(* Logix 5000 project; controller AMP_Servo_Demo vendor 1 type 14 code 154 rev 32.15; software revision 32.05; part 5 of 5 *)
(* tags used below, declared in another part *)
   AMP_Axis1_Absolute_Move_Inst : AMP_Absolute_Move;
   AMP_Axis1_Alarm_Code_Inst : AMP_Alarm_Code;
   AMP_Axis1_Alarm_Reset_Inst : AMP_Alarm_Reset;
   AMP_Axis1_Crash_Stop_Inst : AMP_Crash_Stop;
   AMP_Axis1_DI_Monitor_Inst : AMP_DI_Monitor;
   AMP_Axis1_DO_Control_Inst : AMP_DO_Control;
   AMP_Axis1_Homing_Inst : AMP_Home;
   AMP_Axis1_Inputs : AMP_Input_Assembly_Servo_v2;
   AMP_Axis1_Motor_Disable_Inst : AMP_Motor_Disable;
   AMP_Axis1_Motor_Enable_Inst : AMP_Motor_Enable;
   AMP_Axis1_Motor_Jog_Inst : AMP_Jog_Move;
   AMP_Axis1_Normal_Stop_Inst : AMP_Normal_Stop;
   AMP_Axis1_Point_to_Poinr_IO_Exec : AMP_Point_to_Point_IO;
   AMP_Axis1_Point_to_Point_FC_Exec : AMP_Point_to_Point_FC;
   AMP_Axis1_Q_Segment_Execute_Inst : AMP_Q_Segment_Execute;
   AMP_Axis1_Relative_Move_Inst : AMP_Relative_Move;
   AMP_Axis1_SCL_Inst : AMP_SCL_Command;
   AMP_Axis1_Set_Position_Inst : AMP_Set_Position;
   AMP_Axis1_Status_Code_Inst : AMP_Status_Code;
   AMP_Axis1_Torque_Inst : AMP_Torque_Control;
   AMP_Axis1_Update_Jog_Speed_Inst : AMP_Update_Jog_Speed;
   AMP_Axis2_Absolute_Move_Inst : AMP_Absolute_Move;
   AMP_Axis2_Alarm_Code_Inst : AMP_Alarm_Code;
   AMP_Axis2_Alarm_Reset_Inst : AMP_Alarm_Reset;
   AMP_Axis2_Crash_Stop_Inst : AMP_Crash_Stop;
   AMP_Axis2_DI_Monitor_Inst : AMP_DI_Monitor;
   AMP_Axis2_DO_Control_Inst : AMP_DO_Control;
   AMP_Axis2_Homing_Inst : AMP_Home;
   AMP_Axis2_Inputs : AMP_Input_Assembly_Servo_v2;
   AMP_Axis2_Motor_Disable_Inst : AMP_Motor_Disable;
   AMP_Axis2_Motor_Enable_Inst : AMP_Motor_Enable;
   AMP_Axis2_Motor_Jog_Inst : AMP_Jog_Move;
   AMP_Axis2_Normal_Stop_Inst : AMP_Normal_Stop;
   AMP_Axis2_Point_to_Poinr_IO_Exec : AMP_Point_to_Point_IO;
   AMP_Axis2_Point_to_Point_FC_Exec : AMP_Point_to_Point_FC;
   AMP_Axis2_Q_Segment_Execute_Inst : AMP_Q_Segment_Execute;
   AMP_Axis2_Relative_Move_Inst : AMP_Relative_Move;
   AMP_Axis2_SCL_Inst : AMP_SCL_Command;
   AMP_Axis2_Set_Position_Inst : AMP_Set_Position;
   AMP_Axis2_Status_Code_Inst : AMP_Status_Code;
   AMP_Axis2_Update_Jog_Speed_Inst : AMP_Update_Jog_Speed;
   AMP_Axis2Torque_Inst : AMP_Torque_Control;
   AMP_Input_Axis1_Inst : AMP_Input_Assembly;
   AMP_Input_Axis2_Inst : AMP_Input_Assembly;
(* Explicit_Messages, continued *)

ROUTINE MainRoutine   (* ladder *)
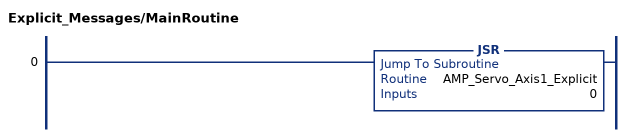
   0: JSR(AMP_Servo_Axis1_Explicit,0);
END_ROUTINE
END_PROGRAM

PROGRAM MainProgram   (* main routine MainRoutine *)

ROUTINE AMP_Servo_Axis1   (* ladder *)
// MDX+ Servo Axis 1 program example using Applied Motion AOIs
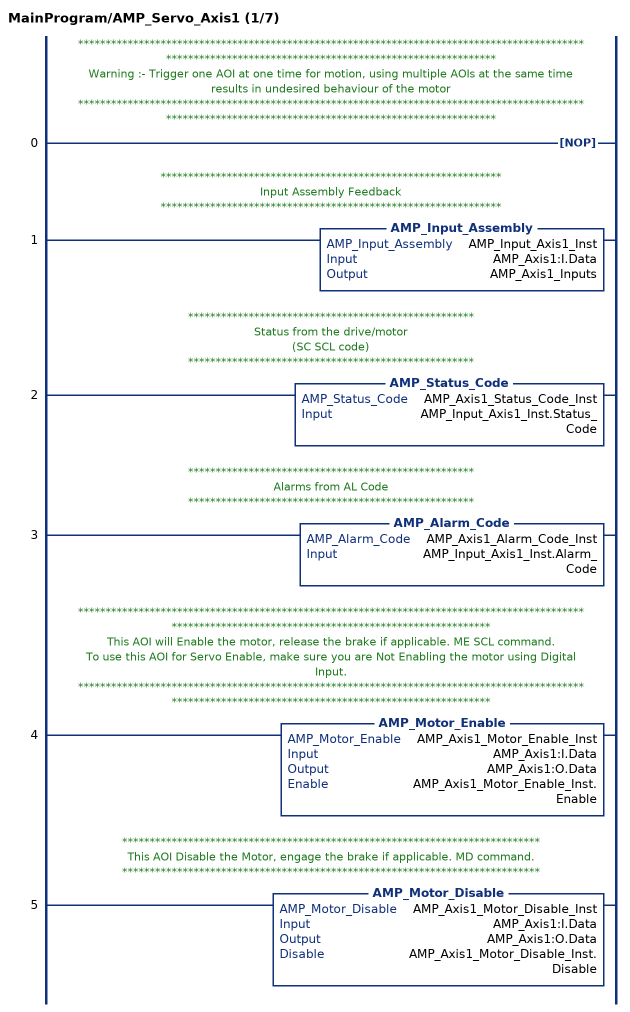
   // ********************************************************************************************************************************************************
   // Warning :- Trigger one AOI at one time for motion, using multiple AOIs at the same time results in undesired behaviour of the motor
   // ********************************************************************************************************************************************************
   0: NOP();
   // **************************************************************
   // Input Assembly Feedback
   // **************************************************************
   1: AMP_Input_Assembly(AMP_Input_Axis1_Inst,AMP_Axis1:I.Data,AMP_Axis1_Inputs);
   // ****************************************************
   // Status from the drive/motor
   // (SC SCL code)
   // ****************************************************
   2: AMP_Status_Code(AMP_Axis1_Status_Code_Inst,AMP_Input_Axis1_Inst.Status_Code);
   // ****************************************************
   //  Alarms from AL Code
   // ****************************************************
   3: AMP_Alarm_Code(AMP_Axis1_Alarm_Code_Inst,AMP_Input_Axis1_Inst.Alarm_Code);
   // ******************************************************************************************************************************************************
   // This AOI will Enable the motor, release the brake if applicable. ME SCL command.
   // To use this AOI for Servo Enable, make sure you are Not Enabling the motor using Digital Input.
   // ******************************************************************************************************************************************************
   4: AMP_Motor_Enable(AMP_Axis1_Motor_Enable_Inst,AMP_Axis1:I.Data,AMP_Axis1:O.Data,AMP_Axis1_Motor_Enable_Inst.Enable);
   // ****************************************************************************
   // This AOI Disable the Motor, engage the brake if applicable. MD command.
   // ****************************************************************************
   5: AMP_Motor_Disable(AMP_Axis1_Motor_Disable_Inst,AMP_Axis1:I.Data,AMP_Axis1:O.Data,AMP_Axis1_Motor_Disable_Inst.Disable);
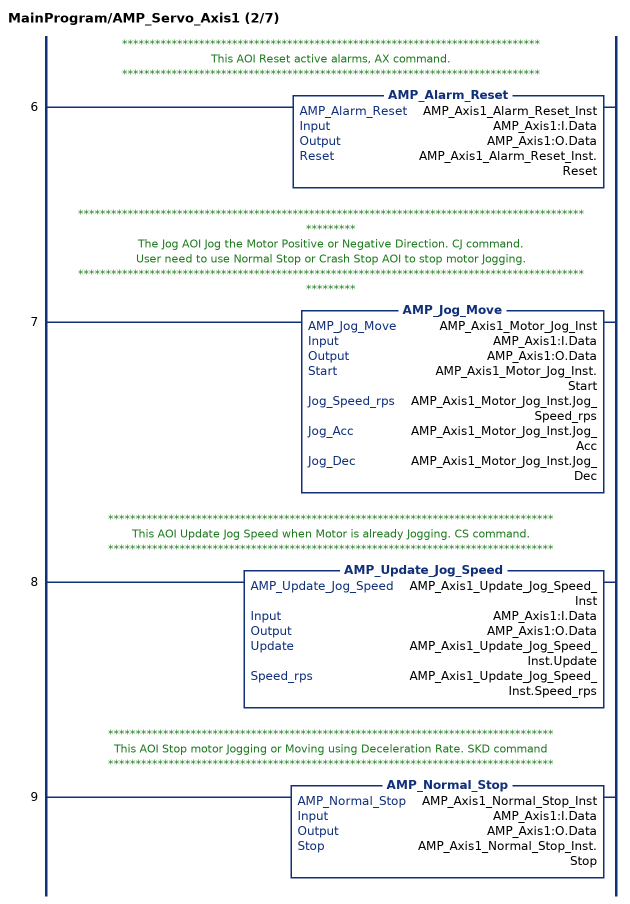
   // ****************************************************************************
   // This AOI Reset active alarms, AX command.
   // ****************************************************************************
   6: AMP_Alarm_Reset(AMP_Axis1_Alarm_Reset_Inst,AMP_Axis1:I.Data,AMP_Axis1:O.Data,AMP_Axis1_Alarm_Reset_Inst.Reset);
   // *****************************************************************************************************
   // The Jog AOI Jog the Motor Positive or Negative Direction. CJ command.
   //  User need to use Normal Stop or Crash Stop AOI to stop motor Jogging.
   // *****************************************************************************************************
   7: AMP_Jog_Move(AMP_Axis1_Motor_Jog_Inst,AMP_Axis1:I.Data,AMP_Axis1:O.Data,AMP_Axis1_Motor_Jog_Inst.Start,AMP_Axis1_Motor_Jog_Inst.Jog_Speed_rps,AMP_Axis1_Motor_Jog_Inst.Jog_Acc,AMP_Axis1_Motor_Jog_Inst.Jog_Dec);
   // *********************************************************************************
   // This AOI Update Jog Speed when Motor is already Jogging. CS command.
   // *********************************************************************************
   8: AMP_Update_Jog_Speed(AMP_Axis1_Update_Jog_Speed_Inst,AMP_Axis1:I.Data,AMP_Axis1:O.Data,AMP_Axis1_Update_Jog_Speed_Inst.Update,AMP_Axis1_Update_Jog_Speed_Inst.Speed_rps);
   // *********************************************************************************
   // This AOI Stop motor Jogging or Moving using Deceleration Rate. SKD command
   // *********************************************************************************
   9: AMP_Normal_Stop(AMP_Axis1_Normal_Stop_Inst,AMP_Axis1:I.Data,AMP_Axis1:O.Data,AMP_Axis1_Normal_Stop_Inst.Stop);
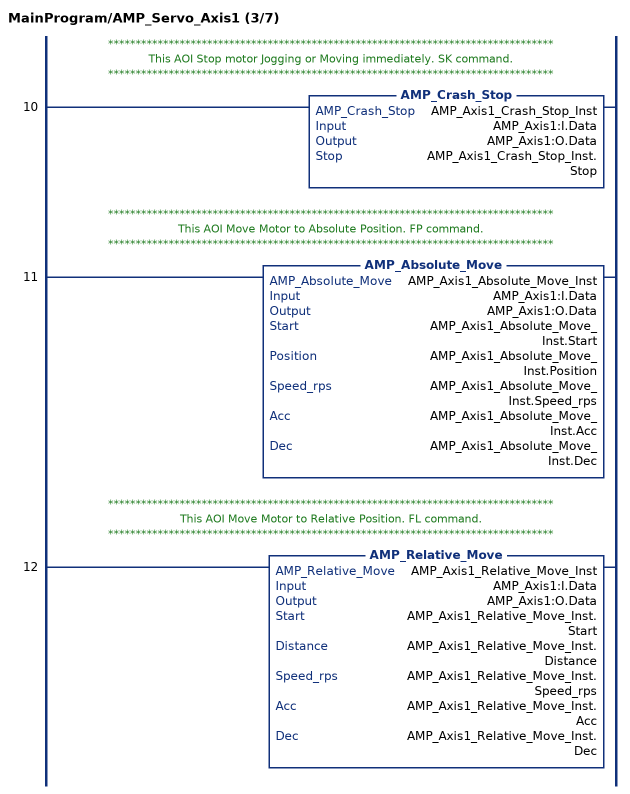
   // *********************************************************************************
   // This AOI Stop motor Jogging or Moving immediately. SK command.
   // *********************************************************************************
   10: AMP_Crash_Stop(AMP_Axis1_Crash_Stop_Inst,AMP_Axis1:I.Data,AMP_Axis1:O.Data,AMP_Axis1_Crash_Stop_Inst.Stop);
   // *********************************************************************************
   // This AOI Move Motor to Absolute Position. FP command.
   // *********************************************************************************
   11: AMP_Absolute_Move(AMP_Axis1_Absolute_Move_Inst,AMP_Axis1:I.Data,AMP_Axis1:O.Data,AMP_Axis1_Absolute_Move_Inst.Start,AMP_Axis1_Absolute_Move_Inst.Position,AMP_Axis1_Absolute_Move_Inst.Speed_rps,AMP_Axis1_Absolute_Move_Inst.Acc,AMP_Axis1_Absolute_Move_Inst.Dec);
   // *********************************************************************************
   // This AOI Move Motor to Relative Position. FL command.
   // *********************************************************************************
   12: AMP_Relative_Move(AMP_Axis1_Relative_Move_Inst,AMP_Axis1:I.Data,AMP_Axis1:O.Data,AMP_Axis1_Relative_Move_Inst.Start,AMP_Axis1_Relative_Move_Inst.Distance,AMP_Axis1_Relative_Move_Inst.Speed_rps,AMP_Axis1_Relative_Move_Inst.Acc,AMP_Axis1_Relative_Move_Inst.Dec);
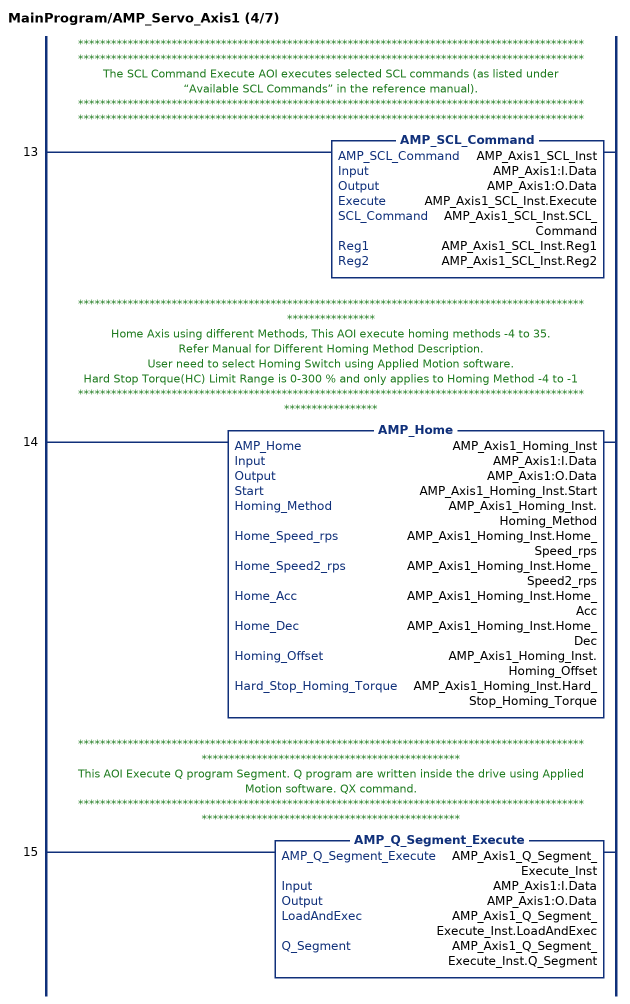
   // ****************************************************************************************************************************************************************************************
   // The SCL Command Execute AOI executes selected SCL commands (as listed under “Available SCL Commands” in the reference manual).
   // ****************************************************************************************************************************************************************************************
   13: AMP_SCL_Command(AMP_Axis1_SCL_Inst,AMP_Axis1:I.Data,AMP_Axis1:O.Data,AMP_Axis1_SCL_Inst.Execute,AMP_Axis1_SCL_Inst.SCL_Command,AMP_Axis1_SCL_Inst.Reg1,AMP_Axis1_SCL_Inst.Reg2);
   // ************************************************************************************************************
   // Home Axis using different Methods, This AOI execute homing methods -4 to 35.
   // Refer Manual for Different Homing Method Description.
   // User need to select Homing Switch using Applied Motion software.
   // Hard Stop Torque(HC) Limit Range is 0-300 % and only applies to Homing Method -4 to -1
   // *************************************************************************************************************
   14: AMP_Home(AMP_Axis1_Homing_Inst,AMP_Axis1:I.Data,AMP_Axis1:O.Data,AMP_Axis1_Homing_Inst.Start,AMP_Axis1_Homing_Inst.Homing_Method,AMP_Axis1_Homing_Inst.Home_Speed_rps,AMP_Axis1_Homing_Inst.Home_Speed2_rps,AMP_Axis1_Homing_Inst.Home_Acc,AMP_Axis1_Homing_Inst.Home_Dec,AMP_Axis1_Homing_Inst.Homing_Offset,AMP_Axis1_Homing_Inst.Hard_Stop_Homing_Torque);
   // *******************************************************************************************************************************************
   // This AOI Execute Q program Segment. Q program are written inside the drive using Applied Motion software. QX command.
   // *******************************************************************************************************************************************
   15: AMP_Q_Segment_Execute(AMP_Axis1_Q_Segment_Execute_Inst,AMP_Axis1:I.Data,AMP_Axis1:O.Data,AMP_Axis1_Q_Segment_Execute_Inst.LoadAndExec,AMP_Axis1_Q_Segment_Execute_Inst.Q_Segment);
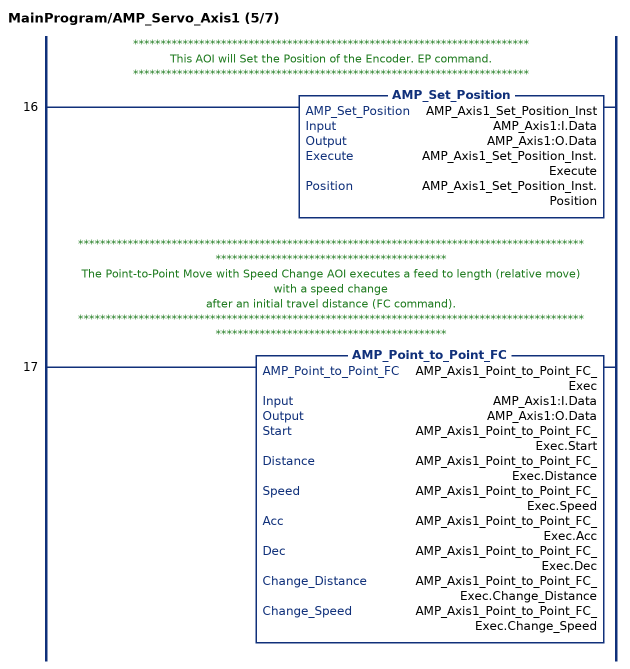
   // ************************************************************************
   // This AOI will Set the Position of the Encoder. EP command.
   // ************************************************************************
   16: AMP_Set_Position(AMP_Axis1_Set_Position_Inst,AMP_Axis1:I.Data,AMP_Axis1:O.Data,AMP_Axis1_Set_Position_Inst.Execute,AMP_Axis1_Set_Position_Inst.Position);
   // **************************************************************************************************************************************
   // The Point-to-Point Move with Speed Change AOI executes a feed to length (relative move) with a speed change
   //  after an initial travel distance (FC command).
   // **************************************************************************************************************************************
   17: AMP_Point_to_Point_FC(AMP_Axis1_Point_to_Point_FC_Exec,AMP_Axis1:I.Data,AMP_Axis1:O.Data,AMP_Axis1_Point_to_Point_FC_Exec.Start,AMP_Axis1_Point_to_Point_FC_Exec.Distance,AMP_Axis1_Point_to_Point_FC_Exec.Speed,AMP_Axis1_Point_to_Point_FC_Exec.Acc,AMP_Axis1_Point_to_Point_FC_Exec.Dec,AMP_Axis1_Point_to_Point_FC_Exec.Change_Distance,AMP_Axis1_Point_to_Point_FC_Exec.Change_Speed);
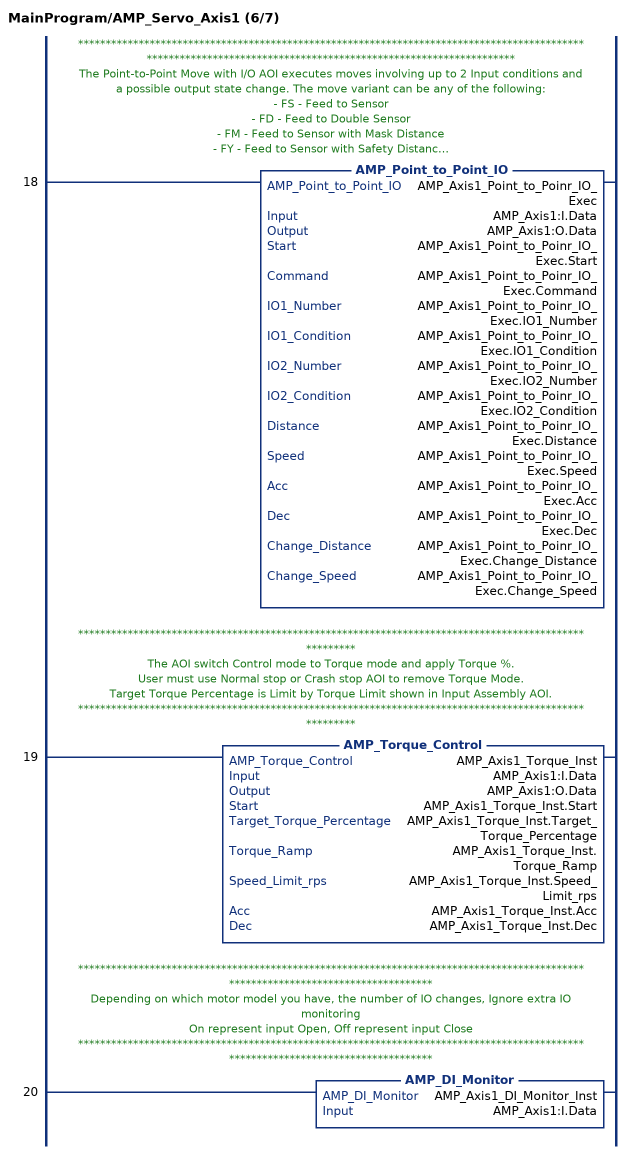
   // ***************************************************************************************************************************************************************
   // The Point-to-Point Move with I/O AOI executes moves involving up to 2 Input conditions and a possible output state change. The move variant can be any of the following:
   // - FS - Feed to Sensor
   // - FD - Feed to Double Sensor
   // - FM - Feed to Sensor with Mask Distance
   // - FY - Feed to Sensor with Safety Distance
   // - FO - Feed to Length and Set Output
   // - SH - Seek Home
   // All six(6) of the above variants need exactly one I/O point except for FD which requires a second I/O point to be specified in the parameters.
   // *************************************************************************************************************************************************************************
   18: AMP_Point_to_Point_IO(AMP_Axis1_Point_to_Poinr_IO_Exec,AMP_Axis1:I.Data,AMP_Axis1:O.Data,AMP_Axis1_Point_to_Poinr_IO_Exec.Start,AMP_Axis1_Point_to_Poinr_IO_Exec.Command,AMP_Axis1_Point_to_Poinr_IO_Exec.IO1_Number,AMP_Axis1_Point_to_Poinr_IO_Exec.IO1_Condition,AMP_Axis1_Point_to_Poinr_IO_Exec.IO2_Number,AMP_Axis1_Point_to_Poinr_IO_Exec.IO2_Condition,AMP_Axis1_Point_to_Poinr_IO_Exec.Distance,AMP_Axis1_Point_to_Poinr_IO_Exec.Speed,AMP_Axis1_Point_to_Poinr_IO_Exec.Acc,AMP_Axis1_Point_to_Poinr_IO_Exec.Dec,AMP_Axis1_Point_to_Poinr_IO_Exec.Change_Distance,AMP_Axis1_Point_to_Poinr_IO_Exec.Change_Speed);
   // *****************************************************************************************************
   // The AOI switch Control mode to Torque mode and apply Torque %.
   // User must use Normal stop or Crash stop AOI to remove Torque Mode.
   // Target Torque Percentage is Limit by Torque Limit shown in Input Assembly AOI.
   // *****************************************************************************************************
   19: AMP_Torque_Control(AMP_Axis1_Torque_Inst,AMP_Axis1:I.Data,AMP_Axis1:O.Data,AMP_Axis1_Torque_Inst.Start,AMP_Axis1_Torque_Inst.Target_Torque_Percentage,AMP_Axis1_Torque_Inst.Torque_Ramp,AMP_Axis1_Torque_Inst.Speed_Limit_rps,AMP_Axis1_Torque_Inst.Acc,AMP_Axis1_Torque_Inst.Dec);
   // *********************************************************************************************************************************
   // Depending on which motor model you have, the number of IO changes, Ignore extra IO monitoring
   // On represent input Open, Off represent input Close
   // *********************************************************************************************************************************
   20: AMP_DI_Monitor(AMP_Axis1_DI_Monitor_Inst,AMP_Axis1:I.Data);
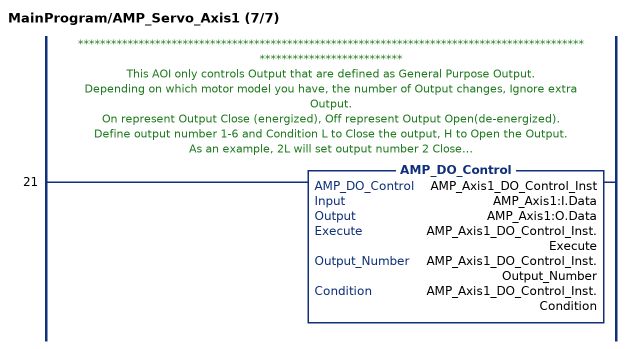
   // **********************************************************************************************************************
   // This AOI only controls Output that are defined as General Purpose Output.
   // Depending on which motor model you have, the number of Output changes, Ignore extra Output.
   // On represent Output Close (energized), Off represent Output Open(de-energized).
   // Define output number 1-6 and Condition L to Close the output, H to Open the Output.
   // As an example, 2L will set output number 2 Close.
   // **********************************************************************************************************************
   21: AMP_DO_Control(AMP_Axis1_DO_Control_Inst,AMP_Axis1:I.Data,AMP_Axis1:O.Data,AMP_Axis1_DO_Control_Inst.Execute,AMP_Axis1_DO_Control_Inst.Output_Number,AMP_Axis1_DO_Control_Inst.Condition);
END_ROUTINE

ROUTINE AMP_Servo_Axis2   (* ladder *)
// M56S Servo Axis 2 program example using Applied Motion AOIs
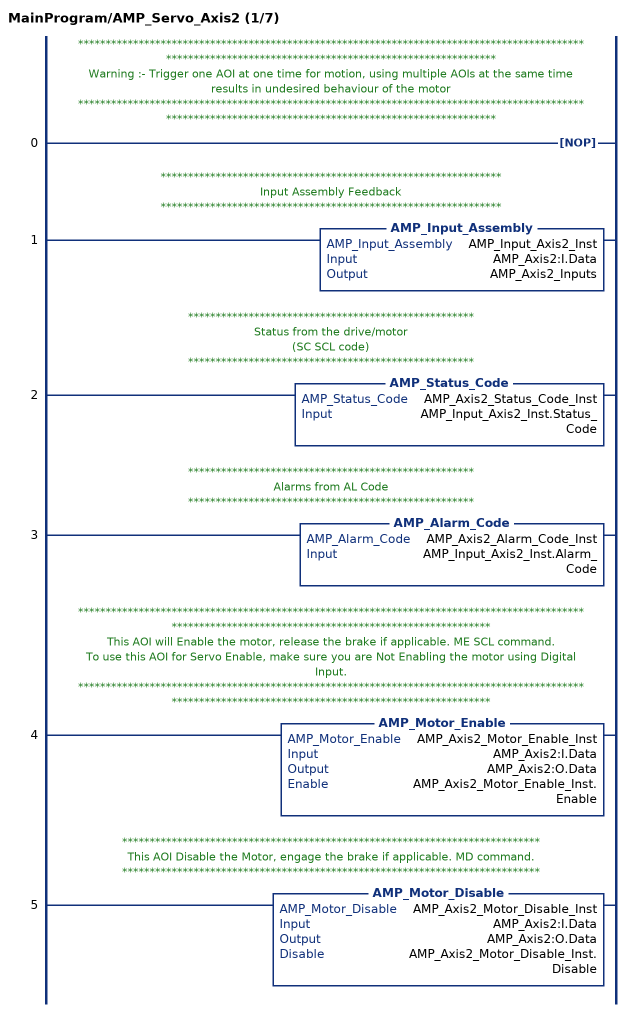
   // ********************************************************************************************************************************************************
   // Warning :- Trigger one AOI at one time for motion, using multiple AOIs at the same time results in undesired behaviour of the motor
   // ********************************************************************************************************************************************************
   0: NOP();
   // **************************************************************
   // Input Assembly Feedback
   // **************************************************************
   1: AMP_Input_Assembly(AMP_Input_Axis2_Inst,AMP_Axis2:I.Data,AMP_Axis2_Inputs);
   // ****************************************************
   // Status from the drive/motor
   // (SC SCL code)
   // ****************************************************
   2: AMP_Status_Code(AMP_Axis2_Status_Code_Inst,AMP_Input_Axis2_Inst.Status_Code);
   // ****************************************************
   //  Alarms from AL Code
   // ****************************************************
   3: AMP_Alarm_Code(AMP_Axis2_Alarm_Code_Inst,AMP_Input_Axis2_Inst.Alarm_Code);
   // ******************************************************************************************************************************************************
   // This AOI will Enable the motor, release the brake if applicable. ME SCL command.
   // To use this AOI for Servo Enable, make sure you are Not Enabling the motor using Digital Input.
   // ******************************************************************************************************************************************************
   4: AMP_Motor_Enable(AMP_Axis2_Motor_Enable_Inst,AMP_Axis2:I.Data,AMP_Axis2:O.Data,AMP_Axis2_Motor_Enable_Inst.Enable);
   // ****************************************************************************
   // This AOI Disable the Motor, engage the brake if applicable. MD command.
   // ****************************************************************************
   5: AMP_Motor_Disable(AMP_Axis2_Motor_Disable_Inst,AMP_Axis2:I.Data,AMP_Axis2:O.Data,AMP_Axis2_Motor_Disable_Inst.Disable);
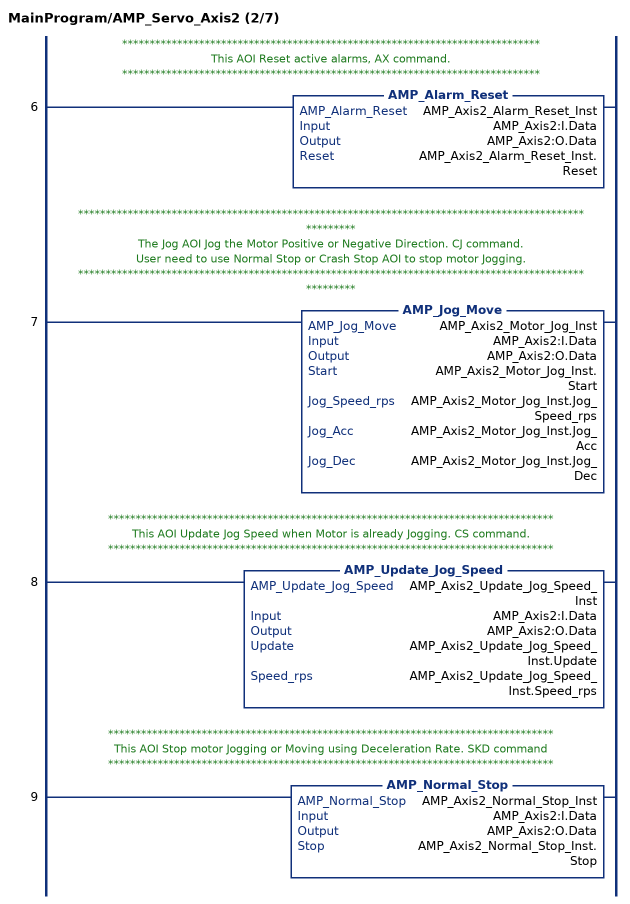
   // ****************************************************************************
   // This AOI Reset active alarms, AX command.
   // ****************************************************************************
   6: AMP_Alarm_Reset(AMP_Axis2_Alarm_Reset_Inst,AMP_Axis2:I.Data,AMP_Axis2:O.Data,AMP_Axis2_Alarm_Reset_Inst.Reset);
   // *****************************************************************************************************
   // The Jog AOI Jog the Motor Positive or Negative Direction. CJ command.
   //  User need to use Normal Stop or Crash Stop AOI to stop motor Jogging.
   // *****************************************************************************************************
   7: AMP_Jog_Move(AMP_Axis2_Motor_Jog_Inst,AMP_Axis2:I.Data,AMP_Axis2:O.Data,AMP_Axis2_Motor_Jog_Inst.Start,AMP_Axis2_Motor_Jog_Inst.Jog_Speed_rps,AMP_Axis2_Motor_Jog_Inst.Jog_Acc,AMP_Axis2_Motor_Jog_Inst.Jog_Dec);
   // *********************************************************************************
   // This AOI Update Jog Speed when Motor is already Jogging. CS command.
   // *********************************************************************************
   8: AMP_Update_Jog_Speed(AMP_Axis2_Update_Jog_Speed_Inst,AMP_Axis2:I.Data,AMP_Axis2:O.Data,AMP_Axis2_Update_Jog_Speed_Inst.Update,AMP_Axis2_Update_Jog_Speed_Inst.Speed_rps);
   // *********************************************************************************
   // This AOI Stop motor Jogging or Moving using Deceleration Rate. SKD command
   // *********************************************************************************
   9: AMP_Normal_Stop(AMP_Axis2_Normal_Stop_Inst,AMP_Axis2:I.Data,AMP_Axis2:O.Data,AMP_Axis2_Normal_Stop_Inst.Stop);
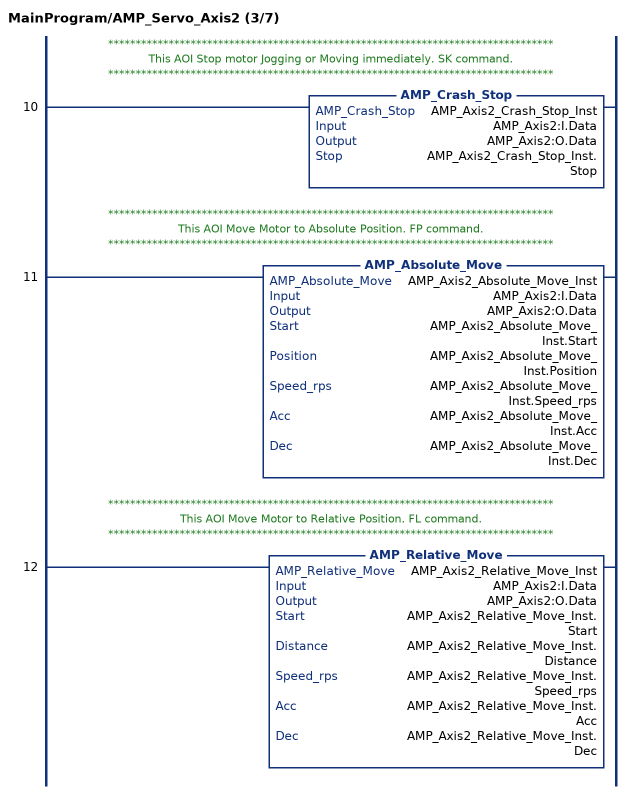
   // *********************************************************************************
   // This AOI Stop motor Jogging or Moving immediately. SK command.
   // *********************************************************************************
   10: AMP_Crash_Stop(AMP_Axis2_Crash_Stop_Inst,AMP_Axis2:I.Data,AMP_Axis2:O.Data,AMP_Axis2_Crash_Stop_Inst.Stop);
   // *********************************************************************************
   // This AOI Move Motor to Absolute Position. FP command.
   // *********************************************************************************
   11: AMP_Absolute_Move(AMP_Axis2_Absolute_Move_Inst,AMP_Axis2:I.Data,AMP_Axis2:O.Data,AMP_Axis2_Absolute_Move_Inst.Start,AMP_Axis2_Absolute_Move_Inst.Position,AMP_Axis2_Absolute_Move_Inst.Speed_rps,AMP_Axis2_Absolute_Move_Inst.Acc,AMP_Axis2_Absolute_Move_Inst.Dec);
   // *********************************************************************************
   // This AOI Move Motor to Relative Position. FL command.
   // *********************************************************************************
   12: AMP_Relative_Move(AMP_Axis2_Relative_Move_Inst,AMP_Axis2:I.Data,AMP_Axis2:O.Data,AMP_Axis2_Relative_Move_Inst.Start,AMP_Axis2_Relative_Move_Inst.Distance,AMP_Axis2_Relative_Move_Inst.Speed_rps,AMP_Axis2_Relative_Move_Inst.Acc,AMP_Axis2_Relative_Move_Inst.Dec);
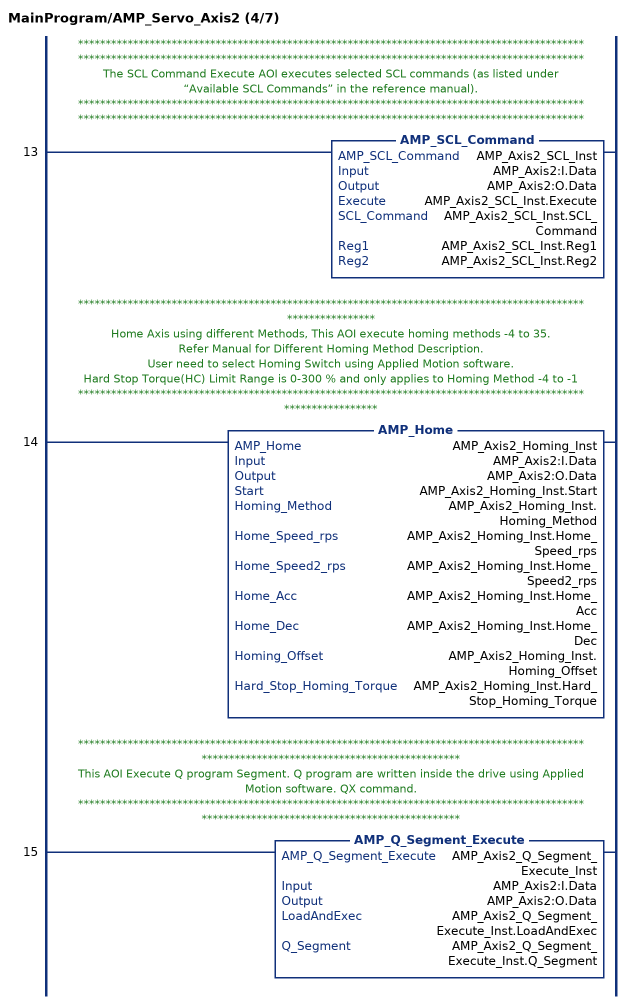
   // ****************************************************************************************************************************************************************************************
   // The SCL Command Execute AOI executes selected SCL commands (as listed under “Available SCL Commands” in the reference manual).
   // ****************************************************************************************************************************************************************************************
   13: AMP_SCL_Command(AMP_Axis2_SCL_Inst,AMP_Axis2:I.Data,AMP_Axis2:O.Data,AMP_Axis2_SCL_Inst.Execute,AMP_Axis2_SCL_Inst.SCL_Command,AMP_Axis2_SCL_Inst.Reg1,AMP_Axis2_SCL_Inst.Reg2);
   // ************************************************************************************************************
   // Home Axis using different Methods, This AOI execute homing methods -4 to 35.
   // Refer Manual for Different Homing Method Description.
   // User need to select Homing Switch using Applied Motion software.
   // Hard Stop Torque(HC) Limit Range is 0-300 % and only applies to Homing Method -4 to -1
   // *************************************************************************************************************
   14: AMP_Home(AMP_Axis2_Homing_Inst,AMP_Axis2:I.Data,AMP_Axis2:O.Data,AMP_Axis2_Homing_Inst.Start,AMP_Axis2_Homing_Inst.Homing_Method,AMP_Axis2_Homing_Inst.Home_Speed_rps,AMP_Axis2_Homing_Inst.Home_Speed2_rps,AMP_Axis2_Homing_Inst.Home_Acc,AMP_Axis2_Homing_Inst.Home_Dec,AMP_Axis2_Homing_Inst.Homing_Offset,AMP_Axis2_Homing_Inst.Hard_Stop_Homing_Torque);
   // *******************************************************************************************************************************************
   // This AOI Execute Q program Segment. Q program are written inside the drive using Applied Motion software. QX command.
   // *******************************************************************************************************************************************
   15: AMP_Q_Segment_Execute(AMP_Axis2_Q_Segment_Execute_Inst,AMP_Axis2:I.Data,AMP_Axis2:O.Data,AMP_Axis2_Q_Segment_Execute_Inst.LoadAndExec,AMP_Axis2_Q_Segment_Execute_Inst.Q_Segment);
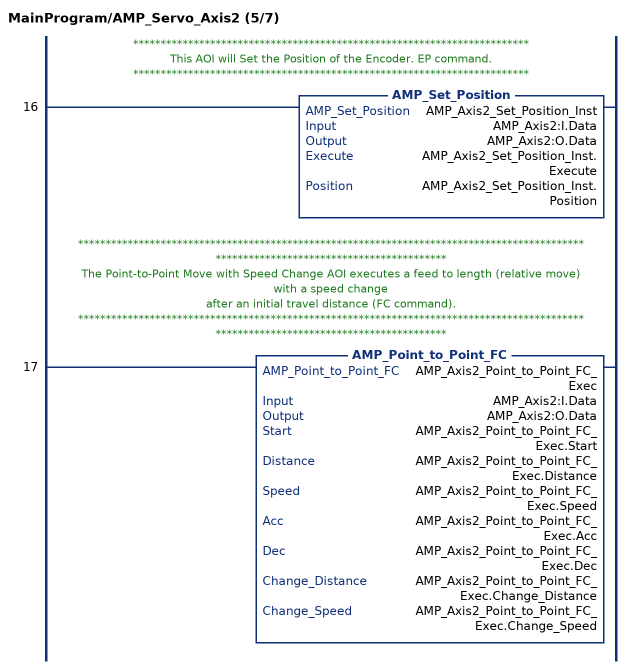
   // ************************************************************************
   // This AOI will Set the Position of the Encoder. EP command.
   // ************************************************************************
   16: AMP_Set_Position(AMP_Axis2_Set_Position_Inst,AMP_Axis2:I.Data,AMP_Axis2:O.Data,AMP_Axis2_Set_Position_Inst.Execute,AMP_Axis2_Set_Position_Inst.Position);
   // **************************************************************************************************************************************
   // The Point-to-Point Move with Speed Change AOI executes a feed to length (relative move) with a speed change
   //  after an initial travel distance (FC command).
   // **************************************************************************************************************************************
   17: AMP_Point_to_Point_FC(AMP_Axis2_Point_to_Point_FC_Exec,AMP_Axis2:I.Data,AMP_Axis2:O.Data,AMP_Axis2_Point_to_Point_FC_Exec.Start,AMP_Axis2_Point_to_Point_FC_Exec.Distance,AMP_Axis2_Point_to_Point_FC_Exec.Speed,AMP_Axis2_Point_to_Point_FC_Exec.Acc,AMP_Axis2_Point_to_Point_FC_Exec.Dec,AMP_Axis2_Point_to_Point_FC_Exec.Change_Distance,AMP_Axis2_Point_to_Point_FC_Exec.Change_Speed);
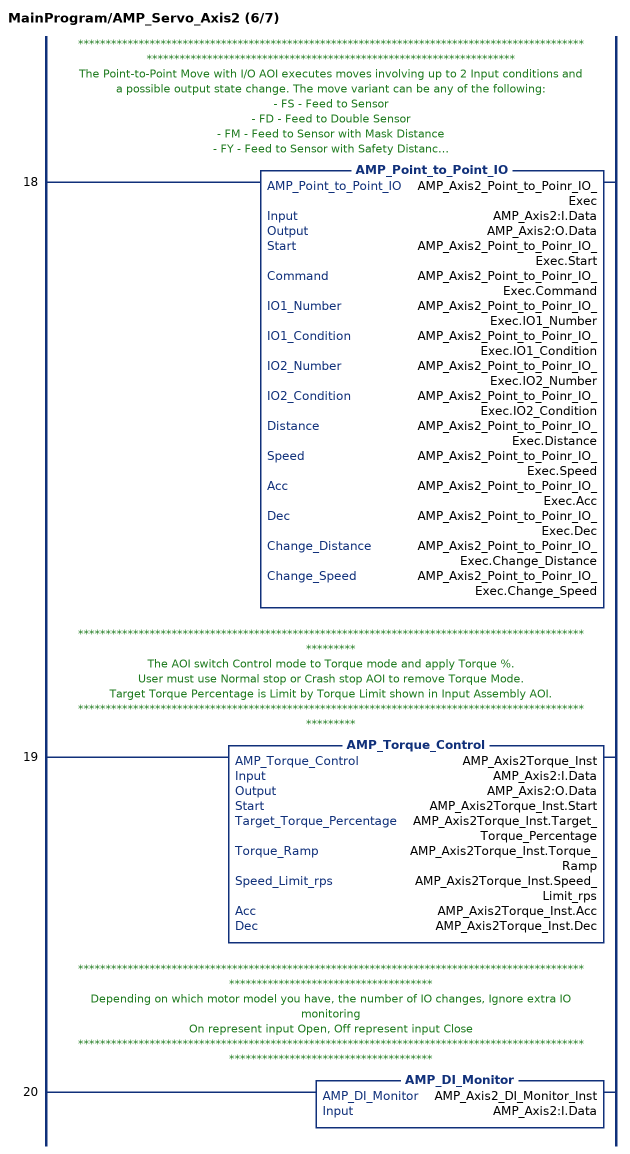
   // ***************************************************************************************************************************************************************
   // The Point-to-Point Move with I/O AOI executes moves involving up to 2 Input conditions and a possible output state change. The move variant can be any of the following:
   // - FS - Feed to Sensor
   // - FD - Feed to Double Sensor
   // - FM - Feed to Sensor with Mask Distance
   // - FY - Feed to Sensor with Safety Distance
   // - FO - Feed to Length and Set Output
   // - SH - Seek Home
   // All six(6) of the above variants need exactly one I/O point except for FD which requires a second I/O point to be specified in the parameters.
   // *************************************************************************************************************************************************************************
   18: AMP_Point_to_Point_IO(AMP_Axis2_Point_to_Poinr_IO_Exec,AMP_Axis2:I.Data,AMP_Axis2:O.Data,AMP_Axis2_Point_to_Poinr_IO_Exec.Start,AMP_Axis2_Point_to_Poinr_IO_Exec.Command,AMP_Axis2_Point_to_Poinr_IO_Exec.IO1_Number,AMP_Axis2_Point_to_Poinr_IO_Exec.IO1_Condition,AMP_Axis2_Point_to_Poinr_IO_Exec.IO2_Number,AMP_Axis2_Point_to_Poinr_IO_Exec.IO2_Condition,AMP_Axis2_Point_to_Poinr_IO_Exec.Distance,AMP_Axis2_Point_to_Poinr_IO_Exec.Speed,AMP_Axis2_Point_to_Poinr_IO_Exec.Acc,AMP_Axis2_Point_to_Poinr_IO_Exec.Dec,AMP_Axis2_Point_to_Poinr_IO_Exec.Change_Distance,AMP_Axis2_Point_to_Poinr_IO_Exec.Change_Speed);
   // *****************************************************************************************************
   // The AOI switch Control mode to Torque mode and apply Torque %.
   // User must use Normal stop or Crash stop AOI to remove Torque Mode.
   // Target Torque Percentage is Limit by Torque Limit shown in Input Assembly AOI.
   // *****************************************************************************************************
   19: AMP_Torque_Control(AMP_Axis2Torque_Inst,AMP_Axis2:I.Data,AMP_Axis2:O.Data,AMP_Axis2Torque_Inst.Start,AMP_Axis2Torque_Inst.Target_Torque_Percentage,AMP_Axis2Torque_Inst.Torque_Ramp,AMP_Axis2Torque_Inst.Speed_Limit_rps,AMP_Axis2Torque_Inst.Acc,AMP_Axis2Torque_Inst.Dec);
   // *********************************************************************************************************************************
   // Depending on which motor model you have, the number of IO changes, Ignore extra IO monitoring
   // On represent input Open, Off represent input Close
   // *********************************************************************************************************************************
   20: AMP_DI_Monitor(AMP_Axis2_DI_Monitor_Inst,AMP_Axis2:I.Data);
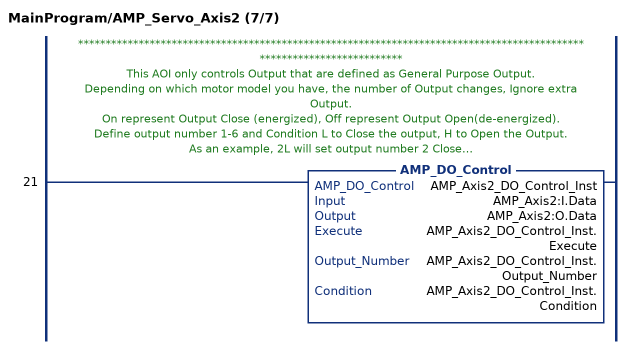
   // **********************************************************************************************************************
   // This AOI only controls Output that are defined as General Purpose Output.
   // Depending on which motor model you have, the number of Output changes, Ignore extra Output.
   // On represent Output Close (energized), Off represent Output Open(de-energized).
   // Define output number 1-6 and Condition L to Close the output, H to Open the Output.
   // As an example, 2L will set output number 2 Close.
   // **********************************************************************************************************************
   21: AMP_DO_Control(AMP_Axis2_DO_Control_Inst,AMP_Axis2:I.Data,AMP_Axis2:O.Data,AMP_Axis2_DO_Control_Inst.Execute,AMP_Axis2_DO_Control_Inst.Output_Number,AMP_Axis2_DO_Control_Inst.Condition);
END_ROUTINE

ROUTINE MainRoutine   (* ladder *)
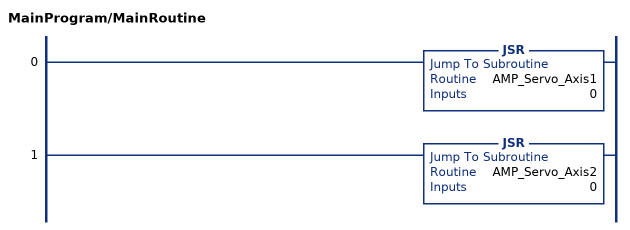
   0: JSR(AMP_Servo_Axis1,0);
   1: JSR(AMP_Servo_Axis2,0);
END_ROUTINE
END_PROGRAM
